/// MODULE INTERFACE INPUT AND OUTPUT 
TYPE DUT_SERVER_MODULE_INTERFACE :
STRUCT
	///Information that the module reads
	Input: DUT_SERVER_MODULE_INTERFACE_INPUT;
	///Information that the module write
	Output: DUT_SERVER_MODULE_INTERFACE_OUTPUT;
END_STRUCT
END_TYPE

(* stored: Version 1.1.0.1, ProductVersion 3.1.0.25
   DUT DUT_SERVER_MODULE_INTERFACE: Id {a0867804-aade-4b4a-ad0c-26a7a1085495} *)
